PROGRAM Stn053_61_Stn231MainMergePrestop
VAR
	{attribute 'TcLinkToOSO' := '.iPuckPresent   :=  <0,1,2>TIIB[N41S00 (AL1332)]^N41S01 (AL2341)^TxPDO^input byte 0;
								 .iBufferFull   :=  <0,1,2>TIIB[N41S00 (AL1332)]^N41S01 (AL2341)^TxPDO^input byte 2;
								 .oStopLower   :=  <0,1,1>TIIB[N41S00 (AL1332)]^N41S02 (EX260)^RxPDO^output byte 0'}
	fbConvStop: FB_ConvStop;
END_VAR

//  This code instantiates a component that is implimented as a common function block
//    Note that I/O is linked directly to I/O variables inside the named instance

gStn053_61_Stn231MainMergePrestop.ConvRunning  := gConsumed_SafetyInterfaceConv.MtrRunning.Enc057Mtr01;

fbConvStop(
	pStn := ADR(gStn053),
	pCmp := ADR(gStn053_61_Stn231MainMergePrestop),
	pUpstreamStop := 0,
	pStateTraceBuffer := ADR(gStn053_StateTraceBuffer),
	pStateTraceFifo := ADR(gStn053_StateTraceFifo),
	pStats := ADR(gStn053_02_Stats));

END_PROGRAM

(* stored: Version 1.1.0.1, ProductVersion 3.1.4024.6
   POU Stn053_61_Stn231MainMergePrestop: Id {ea73f0c0-88d1-4f4e-97f7-a473757c09ca}, SpecialFunc None *)
